SYSTEM TRAFFIC (* System Configuration *)
  (* Standard: 61499-1 *)
  (* Version 0.4, 2009-03-05, JHC, Holobloc Inc., Deleted Application. *)
  (* Version 0.3, 2003-12-05, JHC, Rockwell Automation, Renamed from NEWSYSTEM. *)
  (* Version 0.2, 2002-11-05, JHC, Rockwell Automation, Fixed missing (empty) FBD in Application. *)
  (* Version 0.1, 2002-01-17, JHC, Rockwell Automation, Minor cleanup *)
  (* Version 0.0, 2000-05-27, JHC, Rockwell Automation *)
  DEVICE Device1 : FRAME_DEVICE(BOUNDS := [100,100,300,110])
    RESOURCE Model : PANEL_RESOURCE
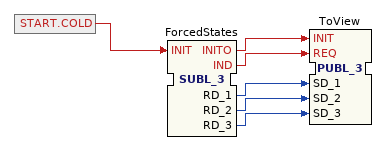
      FBS
        ForcedStates : SUBL_3;
        ToView : PUBL_3;
      END_FBS
      EVENT_CONNECTIONS
        START.COLD TO ForcedStates.INIT;
        ForcedStates.INITO TO ToView.INIT;
        ForcedStates.IND TO ToView.REQ;
      END_CONNECTIONS
      DATA_CONNECTIONS
        ForcedStates.RD_1 TO ToView.SD_1;
        ForcedStates.RD_2 TO ToView.SD_2;
        ForcedStates.RD_3 TO ToView.SD_3;
      END_CONNECTIONS
    END_RESOURCE
    RESOURCE View : PANEL_RESOURCE
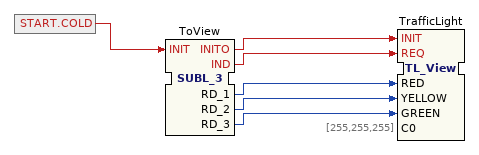
      FBS
        TrafficLight : TL_View(C0 := [255,255,255]);
        ToView : SUBL_3;
      END_FBS
      EVENT_CONNECTIONS
        START.COLD TO ToView.INIT;
        ToView.INITO TO TrafficLight.INIT;
        ToView.IND TO TrafficLight.REQ;
      END_CONNECTIONS
      DATA_CONNECTIONS
        ToView.RD_1 TO TrafficLight.RED;
        ToView.RD_2 TO TrafficLight.YELLOW;
        ToView.RD_3 TO TrafficLight.GREEN;
      END_CONNECTIONS
    END_RESOURCE
    RESOURCE Control : PANEL_RESOURCE
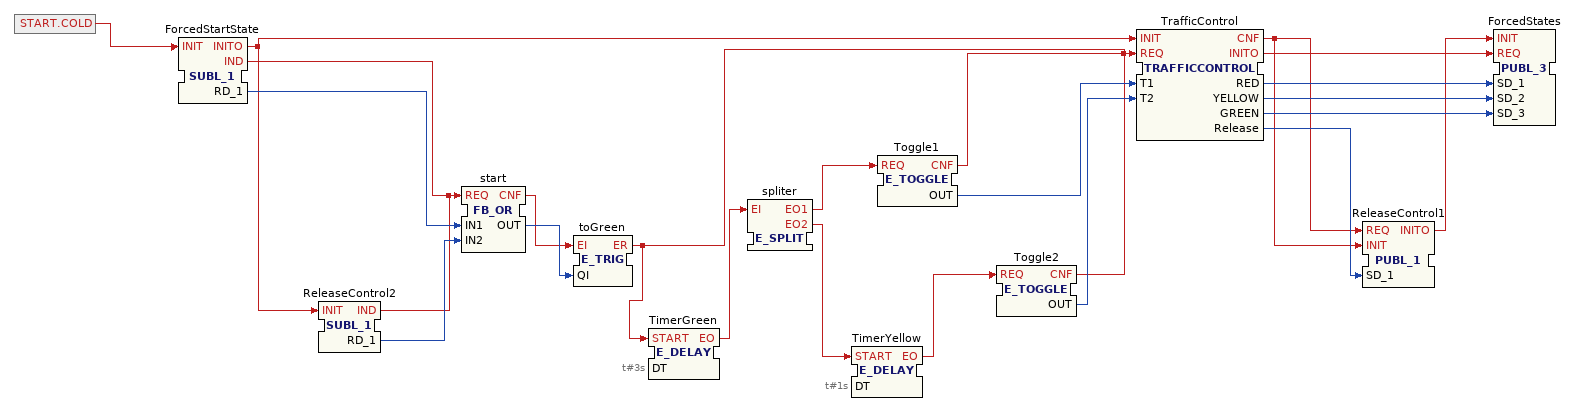
      FBS
        ForcedStartState : SUBL_1;
        spliter : E_SPLIT;
        ForcedStates : PUBL_3;
        TimerGreen : E_DELAY(DT := t#3s);
        Toggle1 : E_TOGGLE;
        Toggle2 : E_TOGGLE;
        TimerYellow : E_DELAY(DT := t#1s);
        ReleaseControl1 : PUBL_1;
        TrafficControl : TRAFFICCONTROL;
        toGreen : E_TRIG;
        start : FB_OR;
        ReleaseControl2 : SUBL_1;
      END_FBS
      EVENT_CONNECTIONS
        START.COLD TO ForcedStartState.INIT;
        TimerGreen.EO TO spliter.EI;
        spliter.EO1 TO Toggle1.REQ;
        spliter.EO2 TO TimerYellow.START;
        ReleaseControl1.INITO TO ForcedStates.INIT;
        ForcedStartState.INITO TO TrafficControl.INIT;
        TrafficControl.CNF TO ForcedStates.REQ;
        TrafficControl.CNF TO ReleaseControl1.REQ;
        TrafficControl.INITO TO ReleaseControl1.INIT;
        Toggle1.CNF TO TrafficControl.REQ;
        Toggle2.CNF TO TrafficControl.REQ;
        TimerYellow.EO TO Toggle2.REQ;
        toGreen.ER TO TimerGreen.START;
        ForcedStartState.IND TO start.REQ;
        start.CNF TO toGreen.EI;
        ForcedStartState.INITO TO ReleaseControl2.INIT;
        ReleaseControl2.IND TO start.REQ;
        toGreen.ER TO TrafficControl.REQ;
      END_CONNECTIONS
      DATA_CONNECTIONS
        TrafficControl.RED TO ForcedStates.SD_1;
        TrafficControl.YELLOW TO ForcedStates.SD_2;
        TrafficControl.GREEN TO ForcedStates.SD_3;
        Toggle1.OUT TO TrafficControl.T1;
        Toggle2.OUT TO TrafficControl.T2;
        TrafficControl.Release TO ReleaseControl1.SD_1;
        start.OUT TO toGreen.QI;
        ForcedStartState.RD_1 TO start.IN1;
        ReleaseControl2.RD_1 TO start.IN2;
      END_CONNECTIONS
    END_RESOURCE
    RESOURCE HMI : PANEL_RESOURCE
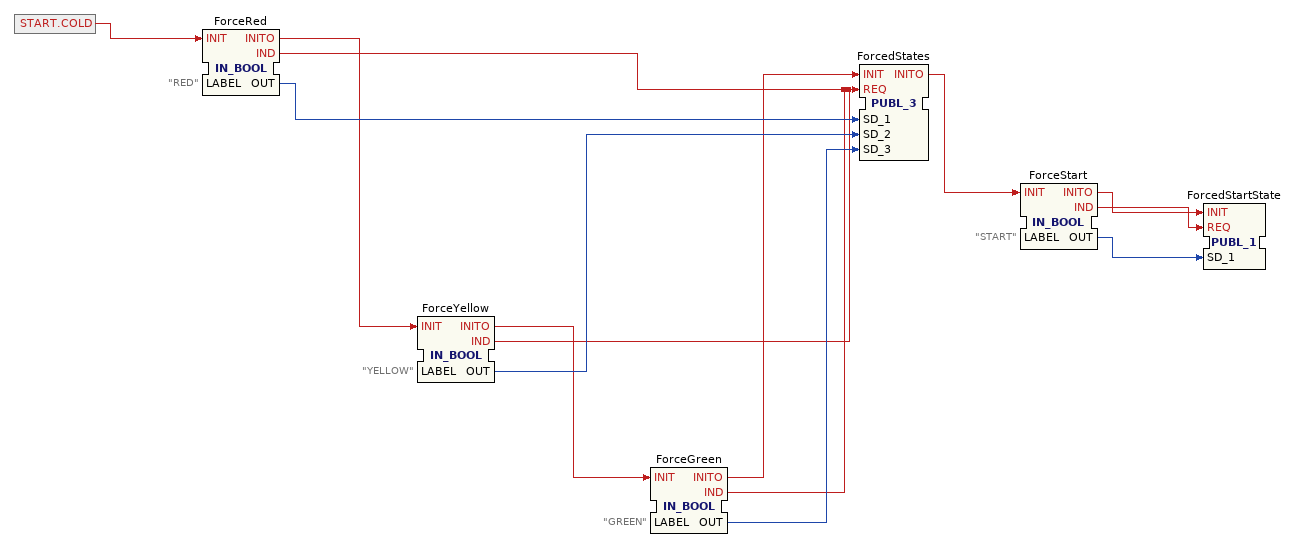
      FBS
        ForceRed : IN_BOOL(LABEL := "RED");
        ForcedStates : PUBL_3;
        ForceYellow : IN_BOOL(LABEL := "YELLOW");
        ForceGreen : IN_BOOL(LABEL := "GREEN");
        ForceStart : IN_BOOL(LABEL := "START");
        ForcedStartState : PUBL_1;
      END_FBS
      EVENT_CONNECTIONS
        START.COLD TO ForceRed.INIT;
        ForceRed.INITO TO ForceYellow.INIT;
        ForceYellow.INITO TO ForceGreen.INIT;
        ForceGreen.INITO TO ForcedStates.INIT;
        ForceRed.IND TO ForcedStates.REQ;
        ForceYellow.IND TO ForcedStates.REQ;
        ForceGreen.IND TO ForcedStates.REQ;
        ForcedStates.INITO TO ForceStart.INIT;
        ForceStart.INITO TO ForcedStartState.INIT;
        ForceStart.IND TO ForcedStartState.REQ;
      END_CONNECTIONS
      DATA_CONNECTIONS
        ForceRed.OUT TO ForcedStates.SD_1;
        ForceYellow.OUT TO ForcedStates.SD_2;
        ForceGreen.OUT TO ForcedStates.SD_3;
        ForceStart.OUT TO ForcedStartState.SD_1;
      END_CONNECTIONS
    END_RESOURCE
  END_DEVICE
  DEVICE Device2 : FRAME_DEVICE(BOUNDS := [100,210,200,110])
    RESOURCE Model : PANEL_RESOURCE
    END_RESOURCE
    RESOURCE View : PANEL_RESOURCE
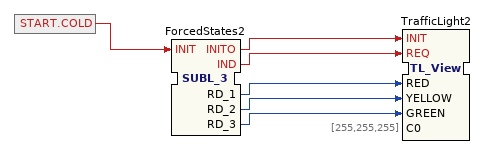
      FBS
        TrafficLight2 : TL_View(C0 := [255,255,255]);
        ForcedStates2 : SUBL_3;
      END_FBS
      EVENT_CONNECTIONS
        START.COLD TO ForcedStates2.INIT;
        ForcedStates2.INITO TO TrafficLight2.INIT;
        ForcedStates2.IND TO TrafficLight2.REQ;
      END_CONNECTIONS
      DATA_CONNECTIONS
        ForcedStates2.RD_1 TO TrafficLight2.RED;
        ForcedStates2.RD_2 TO TrafficLight2.YELLOW;
        ForcedStates2.RD_3 TO TrafficLight2.GREEN;
      END_CONNECTIONS
    END_RESOURCE
    RESOURCE Control : PANEL_RESOURCE
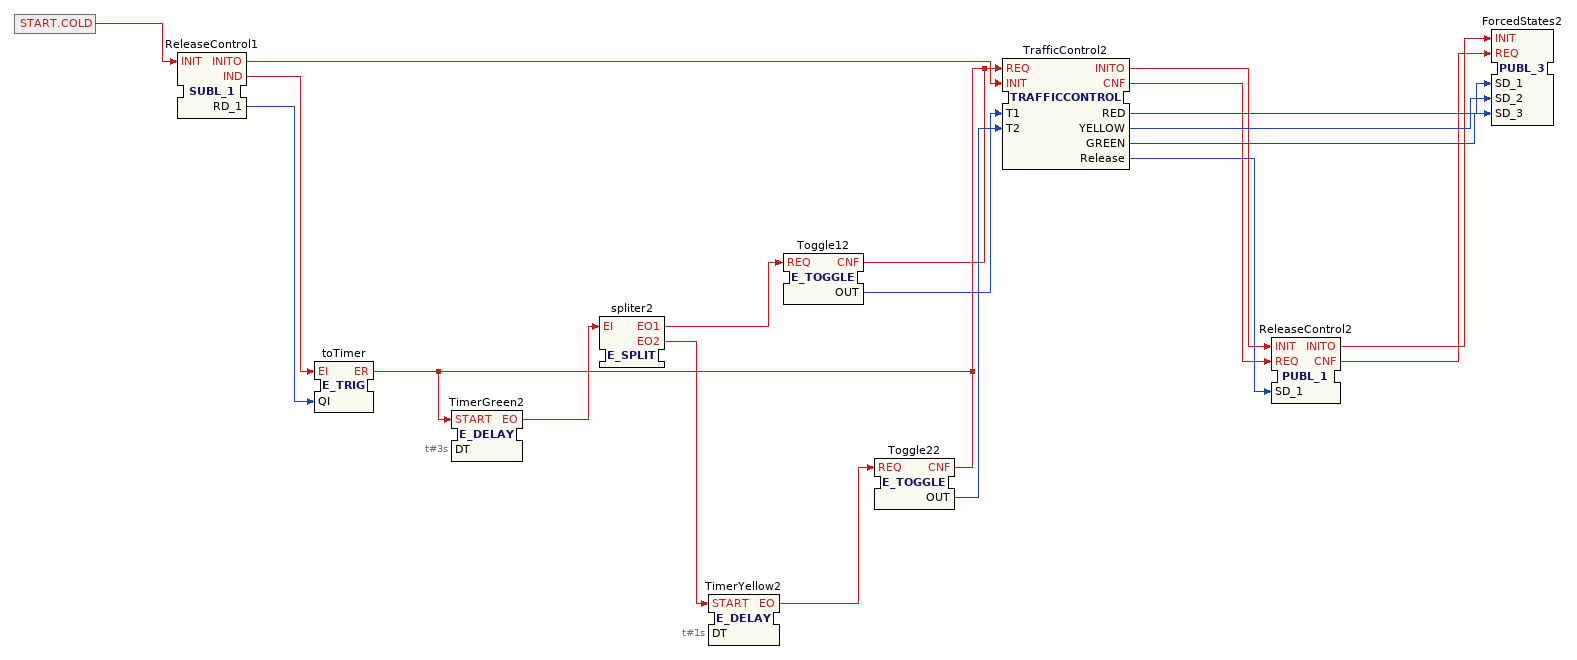
      FBS
        spliter2 : E_SPLIT;
        ForcedStates2 : PUBL_3;
        TimerGreen2 : E_DELAY(DT := t#3s);
        Toggle12 : E_TOGGLE;
        TrafficControl2 : TRAFFICCONTROL;
        Toggle22 : E_TOGGLE;
        TimerYellow2 : E_DELAY(DT := t#1s);
        ReleaseControl1 : SUBL_1;
        toTimer : E_TRIG;
        ReleaseControl2 : PUBL_1;
      END_FBS
      EVENT_CONNECTIONS
        TimerGreen2.EO TO spliter2.EI;
        spliter2.EO1 TO Toggle12.REQ;
        Toggle12.CNF TO TrafficControl2.REQ;
        Toggle22.CNF TO TrafficControl2.REQ;
        spliter2.EO2 TO TimerYellow2.START;
        TimerYellow2.EO TO Toggle22.REQ;
        START.COLD TO ReleaseControl1.INIT;
        ReleaseControl1.INITO TO TrafficControl2.INIT;
        ReleaseControl1.IND TO toTimer.EI;
        toTimer.ER TO TimerGreen2.START;
        toTimer.ER TO TrafficControl2.REQ;
        TrafficControl2.INITO TO ReleaseControl2.INIT;
        TrafficControl2.CNF TO ReleaseControl2.REQ;
        ReleaseControl2.INITO TO ForcedStates2.INIT;
        ReleaseControl2.CNF TO ForcedStates2.REQ;
      END_CONNECTIONS
      DATA_CONNECTIONS
        Toggle12.OUT TO TrafficControl2.T1;
        Toggle22.OUT TO TrafficControl2.T2;
        TrafficControl2.RED TO ForcedStates2.SD_1;
        TrafficControl2.YELLOW TO ForcedStates2.SD_2;
        TrafficControl2.GREEN TO ForcedStates2.SD_3;
        ReleaseControl1.RD_1 TO toTimer.QI;
        TrafficControl2.Release TO ReleaseControl2.SD_1;
      END_CONNECTIONS
    END_RESOURCE
    RESOURCE HMI : PANEL_RESOURCE
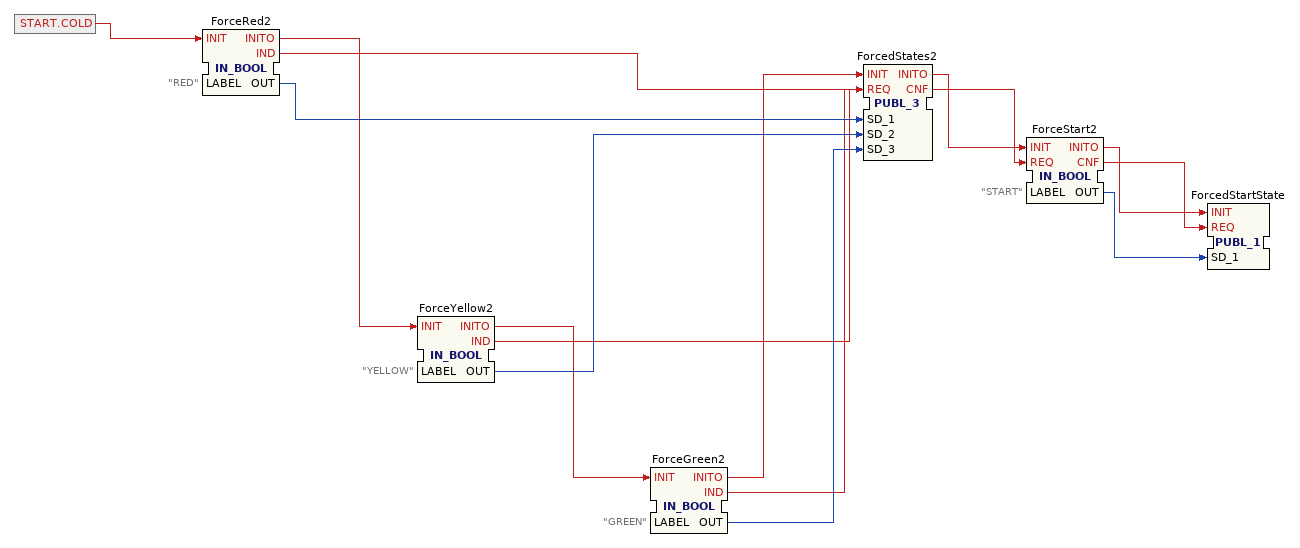
      FBS
        ForceRed2 : IN_BOOL(LABEL := "RED");
        ForcedStates2 : PUBL_3;
        ForceYellow2 : IN_BOOL(LABEL := "YELLOW");
        ForceGreen2 : IN_BOOL(LABEL := "GREEN");
        ForcedStartState : PUBL_1;
        ForceStart2 : IN_BOOL(LABEL := "START");
      END_FBS
      EVENT_CONNECTIONS
        START.COLD TO ForceRed2.INIT;
        ForceRed2.INITO TO ForceYellow2.INIT;
        ForceYellow2.INITO TO ForceGreen2.INIT;
        ForceGreen2.INITO TO ForcedStates2.INIT;
        ForceRed2.IND TO ForcedStates2.REQ;
        ForceYellow2.IND TO ForcedStates2.REQ;
        ForceGreen2.IND TO ForcedStates2.REQ;
        ForcedStates2.INITO TO ForceStart2.INIT;
        ForcedStates2.CNF TO ForceStart2.REQ;
        ForceStart2.INITO TO ForcedStartState.INIT;
        ForceStart2.CNF TO ForcedStartState.REQ;
      END_CONNECTIONS
      DATA_CONNECTIONS
        ForceRed2.OUT TO ForcedStates2.SD_1;
        ForceYellow2.OUT TO ForcedStates2.SD_2;
        ForceGreen2.OUT TO ForcedStates2.SD_3;
        ForceStart2.OUT TO ForcedStartState.SD_1;
      END_CONNECTIONS
    END_RESOURCE
  END_DEVICE
END_SYSTEM
